(* IEC 61131-3 sources: 2026_Projet_YGO_ExcavatriceDragage/CODE/SIMULATION/PLC_TESTS/SUITE_SAFETY, 3 files *)

(* ---- FB_HeartbeatValidation.st ---- *)
(* ═══════════════════════════════════════════════════════════════
   💓 FB_HeartbeatValidation — Suite table-driven Heartbeat IHM↔PLC
   ───────────────────────────────────────────────────────────────
   📄 Doc : DOC/AF_Partie-14_PLC_Tests_Validation_v1.2.md §7
   🎯 Simulation uniquement. Stimuli amont : toggle IHM, demande SEMI_AUTO,
      retours contacteurs/frein M1/M2, frein M3. Jamais d'écriture dans
      SafeStop/PowerCutOff/HeartbeatOk calculés.
   🧪 TC-H1 sain ; TC-H2 perte 2 s ; TC-H3 reprise sans redémarrage ;
      TC-H4 reset conscient ; TC-H5 escalade Méca B M3.
   ═══════════════════════════════════════════════════════════════ *)

FUNCTION_BLOCK PUBLIC FB_HeartbeatValidation
VAR_INPUT
    Start       : BOOL;
    Abort       : BOOL;
    CaseId      : INT; // 0=tous ; 1..5=cas ciblé
END_VAR
VAR_OUTPUT
    Busy                    : BOOL;
    Done                    : BOOL;
    AnyFailed               : BOOL;
    SimGateOk               : BOOL;
    ActiveStimulusId        : INT;
    StepElapsed             : TIME;
    Report                  : ST_TestSuiteReport;
    TerminalState           : E_TestTerminalState;
    ConfigError             : BOOL;
    ConfigErrorStepId       : INT;
    ConfigErrorCheckIdx     : INT;
    ErrorCode               : INT;
    ErrorMessage            : STRING(160);
END_VAR
VAR CONSTANT
    // ── Sondes ──
    SigHeartbeatIhmOk       : INT := 1;
    SigHeartbeatIhmTimeout  : INT := 2;
    SigSafetyM1ErrorId      : INT := 3;
    SigSafetyM2ErrorId      : INT := 4;
    SigSafetyM3ErrorId      : INT := 5;
    SigCycleErrorId         : INT := 6;
    SigM1FwdRevSpeedFbOff   : INT := 7;
    SigM1BrakeFeedback      : INT := 8;
    SigM2FwdRevSpeedFbOff   : INT := 9;
    SigM2BrakeFeedback      : INT := 10;
    SigM3BrakeFeedback      : INT := 11;
    SigM3DriveActualFreqHz  : INT := 12;
    SigM3DriveStatusWord    : INT := 13;
    SigPowerCutOffActive    : INT := 14;
    // ── Étapes ──
    StepTcH1Setup           : INT := 10;
    StepTcH1WaitToggle      : INT := 11;
    StepTcH1Assert          : INT := 12;
    StepTcH1Teardown        : INT := 19;
    StepTcH2Setup           : INT := 20;
    StepTcH2Freeze          : INT := 21;
    StepTcH2Assert          : INT := 22;
    StepTcH2Teardown        : INT := 29;
    StepTcH3Setup           : INT := 30;
    StepTcH3Resume          : INT := 31;
    StepTcH3Assert          : INT := 32;
    StepTcH3Teardown        : INT := 39;
    StepTcH4Setup           : INT := 40;
    StepTcH4Reset           : INT := 41;
    StepTcH4Assert          : INT := 42;
    StepTcH4Teardown        : INT := 49;
    StepTcH5Setup           : INT := 50;
    StepTcH5MecaB           : INT := 51;
    StepTcH5Assert          : INT := 52;
    StepTcH5Teardown        : INT := 59;
END_VAR
VAR
    // Moteur
    Sequencer               : FB_TestSequencer;
    // Tables
    StepTable               : ARRAY[1..GVL_PLC_Tests_Const.MaxSteps]      OF ST_TestStepConfig;
    CheckTable              : ARRAY[1..GVL_PLC_Tests_Const.MaxChecks]     OF ST_TestCheckConfig;
    CaseTable               : ARRAY[1..GVL_PLC_Tests_Const.MaxTestCases]  OF ST_TestCaseConfig;
    InvariantTable          : ARRAY[1..GVL_PLC_Tests_Const.MaxInvariants] OF ST_TestInvariantConfig;
    // Sondes
    ProbeBool               : ARRAY[1..GVL_PLC_Tests_Const.MaxProbeBool]  OF BOOL;
    ProbeDint               : ARRAY[1..GVL_PLC_Tests_Const.MaxProbeDint]  OF DINT;
    ProbeReal               : ARRAY[1..GVL_PLC_Tests_Const.MaxProbeReal]  OF REAL;
    TableReady              : BOOL := FALSE;
    StartPrev               : BOOL;
    // Stimuli locaux
    StimToggleTimer         : TON;
    StimModeRequest         : E_Mode;
    StimResetPulseTimer     : TON;
END_VAR

// ═══════════════════════════════════════════════════════════════
// 1. 🛡️ GATE
// ═══════════════════════════════════════════════════════════════
IF NOT GVL_Simulation.SimulationModeActive THEN
    Sequencer(Start := FALSE, Abort := TRUE, CaseId := CaseId,
              StepTable := StepTable, CheckTable := CheckTable, CaseTable := CaseTable, InvariantTable := InvariantTable,
              ProbeBool := ProbeBool, ProbeDint := ProbeDint, ProbeReal := ProbeReal, Report := Report);
    GVL_PLC_Tests.OverrideIhmHeartbeatActive := FALSE;
    GVL_PLC_Tests.OverrideM3BrakeStuckOpen := FALSE;
    GVL_PLC_Tests.OverrideM1FwdRevSpeedFbOff := FALSE;
    GVL_PLC_Tests.OverrideM1BrakeFeedback := FALSE;
    GVL_PLC_Tests.OverrideM2FwdRevSpeedFbOff := FALSE;
    GVL_PLC_Tests.OverrideM2BrakeFeedback := FALSE;
    GVL_IHM.Modes.BtnFaultReset := FALSE;
    GVL_IHM.Cycle.CmdReset := FALSE;
    Busy := FALSE; Done := TRUE; AnyFailed := TRUE;
    TerminalState := E_TestTerminalState.TEST_TERMINAL_ABORTED;
    Report.InProgress := FALSE; Report.Aborted := TRUE; Report.AnyFailed := TRUE;
    Report.TerminalState := TerminalState; Report.FailureSummary := 'Heartbeat : NOT SimulationModeActive';
    RETURN;
END_IF;

SimGateOk := GVL_Simulation.SimulationModeActive
          AND NOT GVL_Simulation.SensorM1ContactorFeedbackIsReal
          AND NOT GVL_Simulation.SensorM2ContactorFeedbackIsReal
          AND NOT GVL_Simulation.SensorBrakeThermalIsReal
          AND NOT GVL_Simulation.SensorM3ContactorFeedbackIsReal;

IF Abort OR NOT SimGateOk THEN
    GVL_PLC_Tests.OverrideIhmHeartbeatActive := FALSE;
    GVL_PLC_Tests.OverrideM3BrakeStuckOpen := FALSE;
    GVL_PLC_Tests.OverrideM1FwdRevSpeedFbOff := FALSE;
    GVL_PLC_Tests.OverrideM1BrakeFeedback := FALSE;
    GVL_PLC_Tests.OverrideM2FwdRevSpeedFbOff := FALSE;
    GVL_PLC_Tests.OverrideM2BrakeFeedback := FALSE;
    GVL_IHM.Modes.BtnFaultReset := FALSE;
    GVL_IHM.Cycle.CmdReset := FALSE;
    IF Busy THEN GVL_IHM.Modes.SelMode := StimModeRequest; END_IF;
    Busy := FALSE; Done := TRUE; AnyFailed := TRUE;
    TerminalState := E_TestTerminalState.TEST_TERMINAL_ABORTED;
    Report.InProgress := FALSE; Report.Aborted := TRUE; Report.AnyFailed := TRUE;
    Report.TerminalState := TerminalState; Report.FailureSummary := 'Heartbeat : ABORTED or SimGateOk=FALSE';
    RETURN;
END_IF;

IF Start AND NOT StartPrev AND NOT Busy THEN
    StartPrev := TRUE;
    Busy := TRUE; Done := FALSE; AnyFailed := FALSE; ConfigError := FALSE;
    ErrorCode := 0; ErrorMessage := '';
    StepElapsed := T#0s;
    StimModeRequest := GVL_IHM.Modes.SelMode;

    Report.Name := 'Heartbeat Validation';
    Report.InProgress := TRUE; Report.AllPassed := FALSE; Report.AnyFailed := FALSE; Report.Aborted := FALSE;
    Report.TerminalState := E_TestTerminalState.TEST_TERMINAL_NONE;
    Report.ErrorCode := 0; Report.ErrorMessage := ''; Report.FailureSummary := '';
    Report.FailedTestCase := 0; Report.Duration := T#0s;
    Report.RunCounter := Report.RunCounter + 1;
END_IF;
IF NOT Start THEN StartPrev := FALSE; END_IF;

IF NOT Busy THEN RETURN; END_IF;

// ═══════════════════════════════════════════════════════════════
// 2. 📋 TABLES (remplissage unique)
// ═══════════════════════════════════════════════════════════════
IF NOT TableReady THEN
    Report.Name := 'Heartbeat Validation';

    // ── Cas de tests ──
    CaseTable[1].Name := 'TC-H1 Heartbeat sain';      CaseTable[1].FirstStep := StepTcH1Setup;
    CaseTable[2].Name := 'TC-H2 Perte IHM 2s';        CaseTable[2].FirstStep := StepTcH2Setup;
    CaseTable[3].Name := 'TC-H3 Reprise sans redem';  CaseTable[3].FirstStep := StepTcH3Setup;
    CaseTable[4].Name := 'TC-H4 Reset conscient';     CaseTable[4].FirstStep := StepTcH4Setup;
    CaseTable[5].Name := 'TC-H5 Escalade Meca B M3';  CaseTable[5].FirstStep := StepTcH5Setup;

    // ── Checks (index = ligne CheckTable) ──
    // 1: HeartbeatIhmOk = TRUE
    CheckTable[1].Kind := E_TestCheckKind.BOOL_EQUAL;   CheckTable[1].Mode := E_TestCheckMode.CHECK_WAIT_UNTIL;
    CheckTable[1].ProbeIdx := SigHeartbeatIhmOk;        CheckTable[1].ExpectedBool := TRUE;
    // 2: bit0 Safety M1 = 0
    CheckTable[2].Kind := E_TestCheckKind.WORD_MASK_NONE; CheckTable[2].Mode := E_TestCheckMode.CHECK_WAIT_UNTIL;
    CheckTable[2].ProbeIdx := SigSafetyM1ErrorId;        CheckTable[2].Mask := 16#0001;
    // 3: bit0 Safety M2 = 0
    CheckTable[3].Kind := E_TestCheckKind.WORD_MASK_NONE; CheckTable[3].Mode := E_TestCheckMode.CHECK_WAIT_UNTIL;
    CheckTable[3].ProbeIdx := SigSafetyM2ErrorId;        CheckTable[3].Mask := 16#0001;
    // 4: bit0 Safety M3 = 0
    CheckTable[4].Kind := E_TestCheckKind.WORD_MASK_NONE; CheckTable[4].Mode := E_TestCheckMode.CHECK_WAIT_UNTIL;
    CheckTable[4].ProbeIdx := SigSafetyM3ErrorId;        CheckTable[4].Mask := 16#0001;
    // 5: bit5 Cycle = 0
    CheckTable[5].Kind := E_TestCheckKind.WORD_MASK_NONE; CheckTable[5].Mode := E_TestCheckMode.CHECK_WAIT_UNTIL;
    CheckTable[5].ProbeIdx := SigCycleErrorId;           CheckTable[5].Mask := 16#0020;

    // 6: HeartbeatIhmOk = FALSE
    CheckTable[6].Kind := E_TestCheckKind.BOOL_EQUAL;    CheckTable[6].Mode := E_TestCheckMode.CHECK_WAIT_UNTIL;
    CheckTable[6].ProbeIdx := SigHeartbeatIhmOk;         CheckTable[6].ExpectedBool := FALSE;
    // 7: HeartbeatIhmTimeout = TRUE
    CheckTable[7].Kind := E_TestCheckKind.BOOL_EQUAL;    CheckTable[7].Mode := E_TestCheckMode.CHECK_WAIT_UNTIL;
    CheckTable[7].ProbeIdx := SigHeartbeatIhmTimeout;    CheckTable[7].ExpectedBool := TRUE;
    // 8: bit0 Safety M1 = 1
    CheckTable[8].Kind := E_TestCheckKind.WORD_MASK_ANY; CheckTable[8].Mode := E_TestCheckMode.CHECK_WAIT_UNTIL;
    CheckTable[8].ProbeIdx := SigSafetyM1ErrorId;        CheckTable[8].Mask := 16#0001;
    // 9: bit0 Safety M2 = 1
    CheckTable[9].Kind := E_TestCheckKind.WORD_MASK_ANY; CheckTable[9].Mode := E_TestCheckMode.CHECK_WAIT_UNTIL;
    CheckTable[9].ProbeIdx := SigSafetyM2ErrorId;        CheckTable[9].Mask := 16#0001;
    // 10: bit0 Safety M3 = 1
    CheckTable[10].Kind := E_TestCheckKind.WORD_MASK_ANY; CheckTable[10].Mode := E_TestCheckMode.CHECK_WAIT_UNTIL;
    CheckTable[10].ProbeIdx := SigSafetyM3ErrorId;       CheckTable[10].Mask := 16#0001;
    // 11: bit5 Cycle = 1
    CheckTable[11].Kind := E_TestCheckKind.WORD_MASK_ANY; CheckTable[11].Mode := E_TestCheckMode.CHECK_WAIT_UNTIL;
    CheckTable[11].ProbeIdx := SigCycleErrorId;          CheckTable[11].Mask := 16#0020;

    // 12: SafeStop M1 (via Error)
    CheckTable[12].Kind := E_TestCheckKind.BOOL_EQUAL;   CheckTable[12].Mode := E_TestCheckMode.CHECK_WAIT_UNTIL;
    CheckTable[12].ProbeIdx := SigSafetyM1ErrorId;       CheckTable[12].ExpectedBool := TRUE;
    // 13: SafeStop M2
    CheckTable[13].Kind := E_TestCheckKind.BOOL_EQUAL;   CheckTable[13].Mode := E_TestCheckMode.CHECK_WAIT_UNTIL;
    CheckTable[13].ProbeIdx := SigSafetyM2ErrorId;       CheckTable[13].ExpectedBool := TRUE;
    // 14: SafeStop M3
    CheckTable[14].Kind := E_TestCheckKind.BOOL_EQUAL;   CheckTable[14].Mode := E_TestCheckMode.CHECK_WAIT_UNTIL;
    CheckTable[14].ProbeIdx := SigSafetyM3ErrorId;       CheckTable[14].ExpectedBool := TRUE;

    // 15: HeartbeatIhmOk = TRUE (reprise)
    CheckTable[15].Kind := E_TestCheckKind.BOOL_EQUAL;   CheckTable[15].Mode := E_TestCheckMode.CHECK_WAIT_UNTIL;
    CheckTable[15].ProbeIdx := SigHeartbeatIhmOk;        CheckTable[15].ExpectedBool := TRUE;
    // 16-19: bit0 M1/M2/M3 = 1, bit5 Cycle = 1 (mémorisation)
    CheckTable[16].Kind := E_TestCheckKind.WORD_MASK_ANY; CheckTable[16].Mode := E_TestCheckMode.CHECK_WAIT_UNTIL;
    CheckTable[16].ProbeIdx := SigSafetyM1ErrorId;       CheckTable[16].Mask := 16#0001;
    CheckTable[17].Kind := E_TestCheckKind.WORD_MASK_ANY; CheckTable[17].Mode := E_TestCheckMode.CHECK_WAIT_UNTIL;
    CheckTable[17].ProbeIdx := SigSafetyM2ErrorId;       CheckTable[17].Mask := 16#0001;
    CheckTable[18].Kind := E_TestCheckKind.WORD_MASK_ANY; CheckTable[18].Mode := E_TestCheckMode.CHECK_WAIT_UNTIL;
    CheckTable[18].ProbeIdx := SigSafetyM3ErrorId;       CheckTable[18].Mask := 16#0001;
    CheckTable[19].Kind := E_TestCheckKind.WORD_MASK_ANY; CheckTable[19].Mode := E_TestCheckMode.CHECK_WAIT_UNTIL;
    CheckTable[19].ProbeIdx := SigCycleErrorId;          CheckTable[19].Mask := 16#0020;

    // 20: Reset → bit0 M1/M2/M3 = 0, bit5 Cycle = 0
    CheckTable[20].Kind := E_TestCheckKind.WORD_MASK_NONE; CheckTable[20].Mode := E_TestCheckMode.CHECK_WAIT_UNTIL;
    CheckTable[20].ProbeIdx := SigSafetyM1ErrorId;         CheckTable[20].Mask := 16#0001;
    CheckTable[21].Kind := E_TestCheckKind.WORD_MASK_NONE; CheckTable[21].Mode := E_TestCheckMode.CHECK_WAIT_UNTIL;
    CheckTable[21].ProbeIdx := SigSafetyM2ErrorId;         CheckTable[21].Mask := 16#0001;
    CheckTable[22].Kind := E_TestCheckKind.WORD_MASK_NONE; CheckTable[22].Mode := E_TestCheckMode.CHECK_WAIT_UNTIL;
    CheckTable[22].ProbeIdx := SigSafetyM3ErrorId;         CheckTable[22].Mask := 16#0001;
    CheckTable[23].Kind := E_TestCheckKind.WORD_MASK_NONE; CheckTable[23].Mode := E_TestCheckMode.CHECK_WAIT_UNTIL;
    CheckTable[23].ProbeIdx := SigCycleErrorId;            CheckTable[23].Mask := 16#0020;

    // 24: TC-H5 Méca B M3 — PowerCutOffActive = TRUE
    CheckTable[24].Kind := E_TestCheckKind.BOOL_EQUAL;   CheckTable[24].Mode := E_TestCheckMode.CHECK_WAIT_UNTIL;
    CheckTable[24].ProbeIdx := SigPowerCutOffActive;     CheckTable[24].ExpectedBool := TRUE;

    // ── Étapes ──
    // TC-H1
    StepTable[StepTcH1Setup].Name := 'H1 Setup SEMI_AUTO + toggle sain';
    StepTable[StepTcH1Setup].CaseId := 1; StepTable[StepTcH1Setup].StimulusId := 1;
    StepTable[StepTcH1Setup].CheckIdx[1] := 1; StepTable[StepTcH1Setup].CheckIdx[2] := 2;
    StepTable[StepTcH1Setup].CheckIdx[3] := 3; StepTable[StepTcH1Setup].CheckIdx[4] := 4;
    StepTable[StepTcH1Setup].CheckIdx[5] := 5;
    StepTable[StepTcH1Setup].TimeoutPT := T#5s; StepTable[StepTcH1Setup].NextOnPass := StepTcH1WaitToggle;
    StepTable[StepTcH1Setup].NextOnFail := StepTcH1Teardown; StepTable[StepTcH1Setup].FailAction := E_TestFailAction.FAIL_CONTINUE;

    StepTable[StepTcH1WaitToggle].Name := 'H1 Attente 1er front post-boot';
    StepTable[StepTcH1WaitToggle].CaseId := 1; StepTable[StepTcH1WaitToggle].StimulusId := 1;
    StepTable[StepTcH1WaitToggle].CheckIdx[1] := 1;
    StepTable[StepTcH1WaitToggle].TimeoutPT := T#4s; StepTable[StepTcH1WaitToggle].NextOnPass := StepTcH1Assert;
    StepTable[StepTcH1WaitToggle].NextOnFail := StepTcH1Teardown; StepTable[StepTcH1WaitToggle].FailAction := E_TestFailAction.FAIL_CONTINUE;

    StepTable[StepTcH1Assert].Name := 'H1 Assert bit0=0 & bit5=0';
    StepTable[StepTcH1Assert].CaseId := 1; StepTable[StepTcH1Assert].StimulusId := 1;
    StepTable[StepTcH1Assert].CheckIdx[1] := 2; StepTable[StepTcH1Assert].CheckIdx[2] := 3;
    StepTable[StepTcH1Assert].CheckIdx[3] := 4; StepTable[StepTcH1Assert].CheckIdx[4] := 5;
    StepTable[StepTcH1Assert].TimeoutPT := T#2s; StepTable[StepTcH1Assert].NextOnPass := StepTcH1Teardown;
    StepTable[StepTcH1Assert].NextOnFail := StepTcH1Teardown; StepTable[StepTcH1Assert].FailAction := E_TestFailAction.FAIL_CONTINUE;

    StepTable[StepTcH1Teardown].Name := 'H1 Teardown';
    StepTable[StepTcH1Teardown].CaseId := 1; StepTable[StepTcH1Teardown].StimulusId := 0;
    StepTable[StepTcH1Teardown].DwellPT := T#200ms; StepTable[StepTcH1Teardown].TimeoutPT := T#1s;
    StepTable[StepTcH1Teardown].NextOnPass := 0; StepTable[StepTcH1Teardown].NextOnFail := 0;

    // TC-H2
    StepTable[StepTcH2Setup].Name := 'H2 Setup toggle figé';
    StepTable[StepTcH2Setup].CaseId := 2; StepTable[StepTcH2Setup].StimulusId := 2;
    StepTable[StepTcH2Setup].TimeoutPT := T#1s; StepTable[StepTcH2Setup].NextOnPass := StepTcH2Freeze;
    StepTable[StepTcH2Setup].NextOnFail := StepTcH2Teardown; StepTable[StepTcH2Setup].FailAction := E_TestFailAction.FAIL_CONTINUE;

    StepTable[StepTcH2Freeze].Name := 'H2 Figer toggle > 2s timeout';
    StepTable[StepTcH2Freeze].CaseId := 2; StepTable[StepTcH2Freeze].StimulusId := 2;
    StepTable[StepTcH2Freeze].TimeoutPT := T#3s; StepTable[StepTcH2Freeze].NextOnPass := StepTcH2Assert;
    StepTable[StepTcH2Freeze].NextOnFail := StepTcH2Teardown; StepTable[StepTcH2Freeze].FailAction := E_TestFailAction.FAIL_CONTINUE;

    StepTable[StepTcH2Assert].Name := 'H2 Assert bit0=1 & SafeStop';
    StepTable[StepTcH2Assert].CaseId := 2; StepTable[StepTcH2Assert].StimulusId := 2;
    StepTable[StepTcH2Assert].CheckIdx[1] := 6;  StepTable[StepTcH2Assert].CheckIdx[2] := 7;
    StepTable[StepTcH2Assert].CheckIdx[3] := 8;  StepTable[StepTcH2Assert].CheckIdx[4] := 9;
    StepTable[StepTcH2Assert].CheckIdx[5] := 10; StepTable[StepTcH2Assert].CheckIdx[6] := 11;
    StepTable[StepTcH2Assert].CheckIdx[7] := 12; StepTable[StepTcH2Assert].CheckIdx[8] := 13;
    StepTable[StepTcH2Assert].CheckIdx[9] := 14;
    StepTable[StepTcH2Assert].TimeoutPT := T#3s; StepTable[StepTcH2Assert].NextOnPass := StepTcH2Teardown;
    StepTable[StepTcH2Assert].NextOnFail := StepTcH2Teardown; StepTable[StepTcH2Assert].FailAction := E_TestFailAction.FAIL_CONTINUE;

    StepTable[StepTcH2Teardown].Name := 'H2 Teardown';
    StepTable[StepTcH2Teardown].CaseId := 2; StepTable[StepTcH2Teardown].StimulusId := 0;
    StepTable[StepTcH2Teardown].DwellPT := T#200ms; StepTable[StepTcH2Teardown].TimeoutPT := T#1s;
    StepTable[StepTcH2Teardown].NextOnPass := 0; StepTable[StepTcH2Teardown].NextOnFail := 0;

    // TC-H3
    StepTable[StepTcH3Setup].Name := 'H3 Setup reprise toggle';
    StepTable[StepTcH3Setup].CaseId := 3; StepTable[StepTcH3Setup].StimulusId := 3;
    StepTable[StepTcH3Setup].TimeoutPT := T#1s; StepTable[StepTcH3Setup].NextOnPass := StepTcH3Resume;
    StepTable[StepTcH3Setup].NextOnFail := StepTcH3Teardown; StepTable[StepTcH3Setup].FailAction := E_TestFailAction.FAIL_CONTINUE;

    StepTable[StepTcH3Resume].Name := 'H3 Reprise toggle > 2s';
    StepTable[StepTcH3Resume].CaseId := 3; StepTable[StepTcH3Resume].StimulusId := 3;
    StepTable[StepTcH3Resume].TimeoutPT := T#3s; StepTable[StepTcH3Resume].NextOnPass := StepTcH3Assert;
    StepTable[StepTcH3Resume].NextOnFail := StepTcH3Teardown; StepTable[StepTcH3Resume].FailAction := E_TestFailAction.FAIL_CONTINUE;

    StepTable[StepTcH3Assert].Name := 'H3 Assert bit0=1 & bit5=1';
    StepTable[StepTcH3Assert].CaseId := 3; StepTable[StepTcH3Assert].StimulusId := 3;
    StepTable[StepTcH3Assert].CheckIdx[1] := 15; StepTable[StepTcH3Assert].CheckIdx[2] := 16;
    StepTable[StepTcH3Assert].CheckIdx[3] := 17; StepTable[StepTcH3Assert].CheckIdx[4] := 18;
    StepTable[StepTcH3Assert].CheckIdx[5] := 19;
    StepTable[StepTcH3Assert].TimeoutPT := T#3s; StepTable[StepTcH3Assert].NextOnPass := StepTcH3Teardown;
    StepTable[StepTcH3Assert].NextOnFail := StepTcH3Teardown; StepTable[StepTcH3Assert].FailAction := E_TestFailAction.FAIL_CONTINUE;

    StepTable[StepTcH3Teardown].Name := 'H3 Teardown';
    StepTable[StepTcH3Teardown].CaseId := 3; StepTable[StepTcH3Teardown].StimulusId := 0;
    StepTable[StepTcH3Teardown].DwellPT := T#200ms; StepTable[StepTcH3Teardown].TimeoutPT := T#1s;
    StepTable[StepTcH3Teardown].NextOnPass := 0; StepTable[StepTcH3Teardown].NextOnFail := 0;

    // TC-H4
    StepTable[StepTcH4Setup].Name := 'H4 Setup reset pulse';
    StepTable[StepTcH4Setup].CaseId := 4; StepTable[StepTcH4Setup].StimulusId := 4;
    StepTable[StepTcH4Setup].TimeoutPT := T#1s; StepTable[StepTcH4Setup].NextOnPass := StepTcH4Reset;
    StepTable[StepTcH4Setup].NextOnFail := StepTcH4Teardown; StepTable[StepTcH4Setup].FailAction := E_TestFailAction.FAIL_CONTINUE;

    StepTable[StepTcH4Reset].Name := 'H4 Pulse Reset IHM & Cycle';
    StepTable[StepTcH4Reset].CaseId := 4; StepTable[StepTcH4Reset].StimulusId := 4;
    StepTable[StepTcH4Reset].TimeoutPT := T#2s; StepTable[StepTcH4Reset].NextOnPass := StepTcH4Assert;
    StepTable[StepTcH4Reset].NextOnFail := StepTcH4Teardown; StepTable[StepTcH4Reset].FailAction := E_TestFailAction.FAIL_CONTINUE;

    StepTable[StepTcH4Assert].Name := 'H4 Assert bit0=0 & bit5=0';
    StepTable[StepTcH4Assert].CaseId := 4; StepTable[StepTcH4Assert].StimulusId := 1; // retour toggle sain
    StepTable[StepTcH4Assert].CheckIdx[1] := 20; StepTable[StepTcH4Assert].CheckIdx[2] := 21;
    StepTable[StepTcH4Assert].CheckIdx[3] := 22; StepTable[StepTcH4Assert].CheckIdx[4] := 23;
    StepTable[StepTcH4Assert].TimeoutPT := T#3s; StepTable[StepTcH4Assert].NextOnPass := StepTcH4Teardown;
    StepTable[StepTcH4Assert].NextOnFail := StepTcH4Teardown; StepTable[StepTcH4Assert].FailAction := E_TestFailAction.FAIL_CONTINUE;

    StepTable[StepTcH4Teardown].Name := 'H4 Teardown';
    StepTable[StepTcH4Teardown].CaseId := 4; StepTable[StepTcH4Teardown].StimulusId := 0;
    StepTable[StepTcH4Teardown].DwellPT := T#200ms; StepTable[StepTcH4Teardown].TimeoutPT := T#1s;
    StepTable[StepTcH4Teardown].NextOnPass := 0; StepTable[StepTcH4Teardown].NextOnFail := 0;

    // TC-H5
    StepTable[StepTcH5Setup].Name := 'H5 Setup Meca B M3 frein open';
    StepTable[StepTcH5Setup].CaseId := 5; StepTable[StepTcH5Setup].StimulusId := 5;
    StepTable[StepTcH5Setup].TimeoutPT := T#1s; StepTable[StepTcH5Setup].NextOnPass := StepTcH5MecaB;
    StepTable[StepTcH5Setup].NextOnFail := StepTcH5Teardown; StepTable[StepTcH5Setup].FailAction := E_TestFailAction.FAIL_CONTINUE;

    StepTable[StepTcH5MecaB].Name := 'H5 Perte IHM + M3 open > 3s';
    StepTable[StepTcH5MecaB].CaseId := 5; StepTable[StepTcH5MecaB].StimulusId := 5;
    StepTable[StepTcH5MecaB].TimeoutPT := T#7s; StepTable[StepTcH5MecaB].NextOnPass := StepTcH5Assert;
    StepTable[StepTcH5MecaB].NextOnFail := StepTcH5Teardown; StepTable[StepTcH5MecaB].FailAction := E_TestFailAction.FAIL_CONTINUE;

    StepTable[StepTcH5Assert].Name := 'H5 Assert PowerCutOffActive';
    StepTable[StepTcH5Assert].CaseId := 5; StepTable[StepTcH5Assert].StimulusId := 5;
    StepTable[StepTcH5Assert].CheckIdx[1] := 24;
    StepTable[StepTcH5Assert].TimeoutPT := T#3s; StepTable[StepTcH5Assert].NextOnPass := StepTcH5Teardown;
    StepTable[StepTcH5Assert].NextOnFail := StepTcH5Teardown; StepTable[StepTcH5Assert].FailAction := E_TestFailAction.FAIL_CONTINUE;

    StepTable[StepTcH5Teardown].Name := 'H5 Teardown';
    StepTable[StepTcH5Teardown].CaseId := 5; StepTable[StepTcH5Teardown].StimulusId := 0;
    StepTable[StepTcH5Teardown].DwellPT := T#200ms; StepTable[StepTcH5Teardown].TimeoutPT := T#1s;
    StepTable[StepTcH5Teardown].NextOnPass := 0; StepTable[StepTcH5Teardown].NextOnFail := 0;

    TableReady := TRUE;
END_IF;

// ═══════════════════════════════════════════════════════════════
// 3. 📥 ACQUIRE — câblage sondes (1 ligne par signal, pas de logique)
// ═══════════════════════════════════════════════════════════════
ProbeBool[SigHeartbeatIhmOk]       := PRG_01_Diagnostics.instIhmHeartbeat.HeartbeatIhmOk;
ProbeBool[SigHeartbeatIhmTimeout]  := PRG_01_Diagnostics.instIhmHeartbeat.HeartbeatIhmTimeout;
ProbeDint[SigSafetyM1ErrorId]      := WORD_TO_DINT(PRG_03_Safety.instSafetyWinchM1.ErrorId);
ProbeDint[SigSafetyM2ErrorId]      := WORD_TO_DINT(PRG_03_Safety.instSafetyWinchM2.ErrorId);
ProbeDint[SigSafetyM3ErrorId]      := WORD_TO_DINT(PRG_03_Safety.instSafetyTranslationM3.ErrorId);
ProbeDint[SigCycleErrorId]         := WORD_TO_DINT(PRG_05_Cycle.instCycle.ErrorId);
ProbeBool[SigM1FwdRevSpeedFbOff]   := PRG_00_Inputs.M1FwdRevSpeedFeedbackOff;
ProbeBool[SigM1BrakeFeedback]      := PRG_00_Inputs.M1BrakeFeedback;
ProbeBool[SigM2FwdRevSpeedFbOff]   := PRG_00_Inputs.M2FwdRevSpeedFeedbackOff;
ProbeBool[SigM2BrakeFeedback]      := PRG_00_Inputs.M2BrakeFeedback;
ProbeBool[SigM3BrakeFeedback]      := PRG_00_Inputs.M3BrakeFeedback;
ProbeReal[SigM3DriveActualFreqHz]  := UINT_TO_REAL(PRG_00_Inputs.M3_ActualFrequencyHz_Filtered) / 100.0;
ProbeDint[SigM3DriveStatusWord]    := WORD_TO_DINT(PRG_00_Inputs.M3_StatusWord_Filtered);
ProbeBool[SigPowerCutOffActive]    := GVL_IHM.Modes.PowerCutOffActive;

// ═══════════════════════════════════════════════════════════════
// 4. ⚙️ MOTEUR
// ═══════════════════════════════════════════════════════════════
Sequencer(Start := Start, Abort := Abort, CaseId := CaseId,
          StepTable := StepTable, CheckTable := CheckTable, CaseTable := CaseTable, InvariantTable := InvariantTable,
          ProbeBool := ProbeBool, ProbeDint := ProbeDint, ProbeReal := ProbeReal, Report := Report,
          Busy => Busy, Done => Done, AnyFailed => AnyFailed,
          ConfigError => ConfigError, ConfigErrorStepId => ConfigErrorStepId, ConfigErrorCheckIdx => ConfigErrorCheckIdx,
          ActiveStimulusId => ActiveStimulusId, StepElapsed => StepElapsed,
          TerminalState => TerminalState, ErrorCode => ErrorCode, ErrorMessage => ErrorMessage);

// ═══════════════════════════════════════════════════════════════
// 5. ⚡ STIMULI — modèle hybride : TOR état-complet + pulse timer
// ═══════════════════════════════════════════════════════════════
// StimulusId 0 = neutre garanti (tout relâché) — sur Done/Abort par le moteur
GVL_PLC_Tests.OverrideIhmHeartbeatActive := FALSE;
GVL_PLC_Tests.OverrideM3BrakeStuckOpen := FALSE;
GVL_PLC_Tests.OverrideM1FwdRevSpeedFbOff := FALSE;
GVL_PLC_Tests.OverrideM1BrakeFeedback := FALSE;
GVL_PLC_Tests.OverrideM2FwdRevSpeedFbOff := FALSE;
GVL_PLC_Tests.OverrideM2BrakeFeedback := FALSE;
GVL_IHM.Modes.SelMode := StimModeRequest;
GVL_IHM.Modes.BtnFaultReset := FALSE;
GVL_IHM.Cycle.CmdReset := FALSE;

CASE ActiveStimulusId OF
    1: // TC-H1/TC-H4 : toggle sain 500 ms + SEMI_AUTO
        GVL_PLC_Tests.OverrideIhmHeartbeatActive := TRUE;
        GVL_IHM.Modes.SelMode := E_Mode.SEMI_AUTO;
        // Toggle 500 ms
        StimToggleTimer(IN := TRUE, PT := T#500ms);
        IF StimToggleTimer.Q THEN
            GVL_PLC_Tests.OverrideIhmHeartbeatToggle := NOT GVL_PLC_Tests.OverrideIhmHeartbeatToggle;
            StimToggleTimer(IN := FALSE);
        END_IF;

    2: // TC-H2 : toggle figé (perte IHM)
        GVL_PLC_Tests.OverrideIhmHeartbeatActive := TRUE;
        GVL_IHM.Modes.SelMode := E_Mode.SEMI_AUTO;
        // OverrideIhmHeartbeatToggle figé = pas de front

    3: // TC-H3 : reprise toggle sain
        GVL_PLC_Tests.OverrideIhmHeartbeatActive := TRUE;
        GVL_IHM.Modes.SelMode := E_Mode.SEMI_AUTO;
        StimToggleTimer(IN := TRUE, PT := T#500ms);
        IF StimToggleTimer.Q THEN
            GVL_PLC_Tests.OverrideIhmHeartbeatToggle := NOT GVL_PLC_Tests.OverrideIhmHeartbeatToggle;
            StimToggleTimer(IN := FALSE);
        END_IF;

    4: // TC-H4 : pulse reset conscient
        GVL_PLC_Tests.OverrideIhmHeartbeatActive := TRUE;
        GVL_IHM.Modes.SelMode := E_Mode.SEMI_AUTO;
        StimToggleTimer(IN := TRUE, PT := T#500ms);
        IF StimToggleTimer.Q THEN
            GVL_PLC_Tests.OverrideIhmHeartbeatToggle := NOT GVL_PLC_Tests.OverrideIhmHeartbeatToggle;
            StimToggleTimer(IN := FALSE);
        END_IF;
        StimResetPulseTimer(IN := TRUE, PT := T#1500ms);
        IF NOT StimResetPulseTimer.Q THEN
            GVL_IHM.Modes.BtnFaultReset := TRUE;
            GVL_IHM.Cycle.CmdReset := TRUE;
        END_IF;

    5: // TC-H5 : perte IHM + frein M3 desserré → Méca B
        GVL_PLC_Tests.OverrideIhmHeartbeatActive := TRUE;
        GVL_IHM.Modes.SelMode := E_Mode.SEMI_AUTO;
        GVL_PLC_Tests.OverrideM3BrakeStuckOpen := TRUE; // frein M3 desserré
        // Toggle figé = perte IHM
END_CASE;

// ═══════════════════════════════════════════════════════════════
// 6. 🛑 Premier échec → fin explicite, stimuli relâchés, rapport figé
// ═══════════════════════════════════════════════════════════════
IF ErrorCode <> 0 THEN
    GVL_PLC_Tests.OverrideIhmHeartbeatActive := FALSE;
    GVL_PLC_Tests.OverrideM3BrakeStuckOpen := FALSE;
    GVL_PLC_Tests.OverrideM1FwdRevSpeedFbOff := FALSE;
    GVL_PLC_Tests.OverrideM1BrakeFeedback := FALSE;
    GVL_PLC_Tests.OverrideM2FwdRevSpeedFbOff := FALSE;
    GVL_PLC_Tests.OverrideM2BrakeFeedback := FALSE;
    GVL_IHM.Modes.BtnFaultReset := FALSE;
    GVL_IHM.Cycle.CmdReset := FALSE;
    GVL_IHM.Modes.SelMode := StimModeRequest;
    Busy := FALSE; Done := TRUE; AnyFailed := TRUE;
    TerminalState := E_TestTerminalState.TEST_TERMINAL_FAILED;
    Report.InProgress := FALSE; Report.TerminalState := TerminalState;
END_IF;

(* ---- FB_PLC_Tests_Management.st ---- *)
FUNCTION_BLOCK PUBLIC FB_PLC_Tests_Management
VAR_INPUT
    instBucket                : REFERENCE TO FB_Bucket;     // 🆕 Instance benne (pour FB_BucketValidation)
    instWinchM2               : REFERENCE TO FB_Winch;      // 🆕 Instance treuil M2 (pour FB_BucketValidation)
END_VAR
VAR
    // 🧱 Instances de test (1 par suite — ajouter une suite = 1 instance + 1 branche CASE,
    // voir AF_Partie-14 §7.3.4)
    instSafetyValidation      : FB_SafetyValidation;
    instTranslationValidation : FB_TranslationValidation;
    instBucketValidation      : FB_BucketValidation;
    instEncoderValidation     : FB_EncoderValidation;
    instModesValidation       : FB_ModesValidation;
    instHeartbeatValidation   : FB_HeartbeatValidation;

    // Triggers pour IHM tactiles
    RunAllTrig           : R_TRIG;
    AbortTrig            : R_TRIG;
    ClearReportTrig      : R_TRIG;

    // Variables de commande internes
    StartSafety          : BOOL;
    AbortSafety          : BOOL;
    RequestedCaseSafety  : INT;
    StartTranslation     : BOOL;
    AbortTranslation     : BOOL;
    RequestedCaseTranslation : INT; // 🆕 2026-07-22 : CaseId direct (0=toutes,1..6) — JAMAIS de FirstStepId (audit v1.0 C2)
    StartBucket           : BOOL;
    AbortBucket           : BOOL;
    RequestedCaseBucket   : INT;
    StartEncoder          : BOOL;
    AbortEncoder          : BOOL;
    RequestedCaseEncoder  : INT;
    StartModes            : BOOL;
    AbortModes            : BOOL;
    RequestedCaseModes    : INT;
    StartHeartbeat        : BOOL;
    AbortHeartbeat        : BOOL;
    RequestedCaseHeartbeat : INT;
    StartFramework        : BOOL;
    FrameworkScanCount    : INT;

    // 🔗 Enchaînement multi-suites (CmdRunAll) — 2026-07-16 : ajout Translation puis Bucket
    ChainMode            : BOOL;  // TRUE = run déclenché par RunAll, enchaîne Safety PUIS Translation PUIS Bucket
    CurrentSuiteIdx      : INT;   // Suite active/dernière active (GVL_PLC_Tests_Const.SuiteSafety/SuiteTranslation/SuiteBucket)
    FinalAborted         : BOOL;
    FinalAnyFailed       : BOOL;
    SuiteElapsed         : TIME;
    SuiteWatchdogExpired : BOOL;
    LastLoggedSafetyRun  : UDINT;
    LastLoggedTranslationRun : UDINT;
    LastLoggedBucketRun  : UDINT;
    LastLoggedHeartbeatRun : UDINT;
    EventIdx             : INT;

    // Compteurs pour progression IHM
    Idx                  : INT;
    PassedCount          : INT;
    FailedCount          : INT;
    TotalCount           : INT;

    // 💓 Gestion du clignotant HMI
    LastStepId           : INT := 0;
    PulseCounter         : INT := 0;
    CycleCounter         : INT := 0;
END_VAR
// === IMPLEMENTATION ===
// 1. Détection des commandes HMI
RunAllTrig(CLK := GVL_PLC_Tests.Cmd.RunAll);
AbortTrig(CLK := GVL_PLC_Tests.Cmd.Abort);
ClearReportTrig(CLK := GVL_PLC_Tests.Cmd.ClearReport);

// Remise à zéro des boutons poussoirs HMI
// 🔧 REX 2026-07-16 (demande utilisateur) : CmdRunAll n'est PAS remis à FALSE ici (contrairement
// à l'ancien CmdRunTests, pulse consommé au scan suivant) — il reste TRUE tout le temps du run,
// pratique pour observer en Watch/forçage CODESYS, et ne retombe qu'au Done (cf. CASE ci-dessous).
// R_TRIG garantit qu'un niveau maintenu ne redéclenche pas un 2e run.
IF GVL_PLC_Tests.Cmd.Abort THEN
    GVL_PLC_Tests.Cmd.Abort := FALSE;
END_IF;
IF GVL_PLC_Tests.Cmd.ClearReport THEN
    GVL_PLC_Tests.Cmd.ClearReport := FALSE;
END_IF;

// 2. Machine d'états principale
CASE GVL_PLC_Tests.Status.RunState OF

    // 🔧 REX 2026-07-16 (demande utilisateur) : PASSED/FAILED/ABORTED sont FIGÉS ici (pattern
    // StateAtError, P3 §4) — sans ça, l'état ne durait qu'1 scan (10ms) avant de retomber tout
    // seul à IDLE, invisible en Watch CODESYS. On ne quitte cet état que sur nouveau Start
    // (relance direct un run) ou CmdClearReport (acquittement explicite → retour IDLE).
    E_TestRunState.TESTRUN_IDLE, E_TestRunState.TESTRUN_PASSED, E_TestRunState.TESTRUN_FAILED, E_TestRunState.TESTRUN_ABORTED:
        StartSafety := FALSE;
        AbortSafety := FALSE;
        StartTranslation := FALSE;
        AbortTranslation := FALSE;
        StartBucket := FALSE;
        AbortBucket := FALSE;
        StartEncoder := FALSE;
        AbortEncoder := FALSE;
        StartModes := FALSE;
        AbortModes := FALSE;
        StartHeartbeat := FALSE;
        AbortHeartbeat := FALSE;
        StartFramework := FALSE;
        SuiteElapsed := T#0s;
        SuiteWatchdogExpired := FALSE;

        // 🧪 RunAll prioritaire : démarre une campagne complète depuis Safety.
        IF RunAllTrig.Q THEN
            ChainMode := TRUE;
            CurrentSuiteIdx := GVL_PLC_Tests_Const.SuiteSafety;
            RequestedCaseSafety := 0;
            RequestedCaseTranslation := 0;
            RequestedCaseBucket := 0;
            RequestedCaseEncoder := 0;
            RequestedCaseModes := 0;
            RequestedCaseHeartbeat := 0;
            FinalAborted := FALSE;
            FinalAnyFailed := FALSE;
            GVL_PLC_Tests.Cmd.RunSuite := 0;
            GVL_PLC_Tests.Cmd.RunCase := 0;
            GVL_PLC_Tests.Status.FailureSummary := '';
            StartSafety := TRUE;
            GVL_PLC_Tests.Status.RunState := E_TestRunState.TESTRUN_RUNNING;
        // Normalisation des commandes unitaires vers RunSuite.
        ELSIF GVL_PLC_Tests.Cmd.RunSafety THEN
            GVL_PLC_Tests.Cmd.RunSuite := GVL_PLC_Tests_Const.SuiteSafety;
            GVL_PLC_Tests.Cmd.RunSafety := FALSE;
        ELSIF GVL_PLC_Tests.Cmd.RunTranslation THEN
            GVL_PLC_Tests.Cmd.RunSuite := GVL_PLC_Tests_Const.SuiteTranslation;
            GVL_PLC_Tests.Cmd.RunTranslation := FALSE;
        ELSIF GVL_PLC_Tests.Cmd.RunBucket THEN
            GVL_PLC_Tests.Cmd.RunSuite := GVL_PLC_Tests_Const.SuiteBucket;
            GVL_PLC_Tests.Cmd.RunBucket := FALSE;
        ELSIF GVL_PLC_Tests.Cmd.RunEncoder THEN
            GVL_PLC_Tests.Cmd.RunSuite := GVL_PLC_Tests_Const.SuiteEncoder;
            GVL_PLC_Tests.Cmd.RunEncoder := FALSE;
        ELSIF GVL_PLC_Tests.Cmd.RunModes THEN
            GVL_PLC_Tests.Cmd.RunSuite := GVL_PLC_Tests_Const.SuiteModes;
            GVL_PLC_Tests.Cmd.RunModes := FALSE;
        ELSIF GVL_PLC_Tests.Cmd.RunHeartbeat THEN
            GVL_PLC_Tests.Cmd.RunSuite := GVL_PLC_Tests_Const.SuiteHeartbeat;
            GVL_PLC_Tests.Cmd.RunHeartbeat := FALSE;
        ELSIF GVL_PLC_Tests.Cmd.RunFramework THEN
            StartFramework := TRUE;
            GVL_PLC_Tests.Cmd.RunFramework := FALSE;
        END_IF;

        // Démarrage d'une suite ciblée (Safety)
        IF GVL_PLC_Tests.Cmd.RunSuite = GVL_PLC_Tests_Const.SuiteSafety THEN
            IF GVL_Simulation.SimulationModeActive AND instSafetyValidation.SimGateOk THEN
                ChainMode := FALSE;
                CurrentSuiteIdx := GVL_PLC_Tests_Const.SuiteSafety;
                StartSafety := TRUE;
                RequestedCaseSafety := GVL_PLC_Tests.Cmd.RunCase;
                GVL_PLC_Tests.Status.FailureSummary := ''; // 🔄 RAZ à chaque nouveau run
                GVL_PLC_Tests.Status.RunState := E_TestRunState.TESTRUN_RUNNING;
            END_IF;
            GVL_PLC_Tests.Cmd.RunSuite := 0;
            GVL_PLC_Tests.Cmd.RunCase := 0;

        // Démarrage d'une suite ciblée (Translation)
        // 🆕 2026-07-22 : CaseId transmis TEL QUEL (0=toutes,1..6) — le manager ne
        // connaît plus aucun détail interne d'étape (audit v1.0 C2). Refus de
        // gate désormais explicite PRECONDITION_FAILED, jamais silencieux (C3).
        ELSIF GVL_PLC_Tests.Cmd.RunSuite = GVL_PLC_Tests_Const.SuiteTranslation THEN
            // La suite possède seule sa fixture : même un refus produit un rapport neuf
            // PRECONDITION_FAILED, jamais un Status correct avec un ancien rapport.
            ChainMode := FALSE;
            CurrentSuiteIdx := GVL_PLC_Tests_Const.SuiteTranslation;
            StartTranslation := TRUE;
            RequestedCaseTranslation := GVL_PLC_Tests.Cmd.RunCase;
            GVL_PLC_Tests.Status.FailureSummary := '';
            GVL_PLC_Tests.Status.RunState := E_TestRunState.TESTRUN_RUNNING;
            GVL_PLC_Tests.Cmd.RunSuite := 0;
            GVL_PLC_Tests.Cmd.RunCase := 0;

        // Démarrage d'une suite ciblée (Bucket)
        ELSIF GVL_PLC_Tests.Cmd.RunSuite = GVL_PLC_Tests_Const.SuiteBucket THEN
            IF GVL_Simulation.SimulationModeActive AND instBucketValidation.SimGateOk THEN
                ChainMode := FALSE;
                CurrentSuiteIdx := GVL_PLC_Tests_Const.SuiteBucket;
                StartBucket := TRUE;
                RequestedCaseBucket := GVL_PLC_Tests.Cmd.RunCase;
                GVL_PLC_Tests.Status.FailureSummary := ''; // 🔄 RAZ à chaque nouveau run
                GVL_PLC_Tests.Status.RunState := E_TestRunState.TESTRUN_RUNNING;
            END_IF;
            GVL_PLC_Tests.Cmd.RunSuite := 0;
            GVL_PLC_Tests.Cmd.RunCase := 0;

        // Démarrage d'une suite ciblée (Codeurs/Homing nominal)
        ELSIF GVL_PLC_Tests.Cmd.RunSuite = GVL_PLC_Tests_Const.SuiteEncoder THEN
            IF GVL_Simulation.SimulationModeActive AND instEncoderValidation.SimGateOk THEN
                ChainMode := FALSE;
                CurrentSuiteIdx := GVL_PLC_Tests_Const.SuiteEncoder;
                StartEncoder := TRUE;
                RequestedCaseEncoder := GVL_PLC_Tests.Cmd.RunCase;
                GVL_PLC_Tests.Status.FailureSummary := '';
                GVL_PLC_Tests.Status.RunState := E_TestRunState.TESTRUN_RUNNING;
            END_IF;
            GVL_PLC_Tests.Cmd.RunSuite := 0;
            GVL_PLC_Tests.Cmd.RunCase := 0;

        // Démarrage d'une suite ciblée (Modes/Homme-mort, post-suppression IHM_MANU)
        ELSIF GVL_PLC_Tests.Cmd.RunSuite = GVL_PLC_Tests_Const.SuiteModes THEN
            IF GVL_Simulation.SimulationModeActive AND instModesValidation.SimGateOk THEN
                ChainMode := FALSE;
                CurrentSuiteIdx := GVL_PLC_Tests_Const.SuiteModes;
                StartModes := TRUE;
                RequestedCaseModes := GVL_PLC_Tests.Cmd.RunCase;
                GVL_PLC_Tests.Status.FailureSummary := '';
                GVL_PLC_Tests.Status.RunState := E_TestRunState.TESTRUN_RUNNING;
            END_IF;
            GVL_PLC_Tests.Cmd.RunSuite := 0;
            GVL_PLC_Tests.Cmd.RunCase := 0;

        // Démarrage suite Heartbeat IHM↔PLC.
        ELSIF GVL_PLC_Tests.Cmd.RunSuite = GVL_PLC_Tests_Const.SuiteHeartbeat THEN
            IF GVL_Simulation.SimulationModeActive
               AND NOT GVL_Simulation.SensorM1ContactorFeedbackIsReal
               AND NOT GVL_Simulation.SensorM2ContactorFeedbackIsReal THEN
                ChainMode := FALSE;
                CurrentSuiteIdx := GVL_PLC_Tests_Const.SuiteHeartbeat;
                StartHeartbeat := TRUE;
                RequestedCaseHeartbeat := GVL_PLC_Tests.Cmd.RunCase;
                GVL_PLC_Tests.Status.FailureSummary := '';
                GVL_PLC_Tests.Status.RunState := E_TestRunState.TESTRUN_RUNNING;
            END_IF;
            GVL_PLC_Tests.Cmd.RunSuite := 0;
            GVL_PLC_Tests.Cmd.RunCase := 0;
        END_IF;

        // 🧪 Smoke test géré directement ici : aucune instance/table/runtime.
        IF StartFramework THEN
            ChainMode := FALSE;
            FrameworkScanCount := 0;
            GVL_PLC_Tests.FrameworkResult.InProgress := TRUE;
            GVL_PLC_Tests.FrameworkResult.AllPassed := FALSE;
            GVL_PLC_Tests.FrameworkResult.AnyFailed := FALSE;
            GVL_PLC_Tests.FrameworkResult.CurrentTestId := 1;
            GVL_PLC_Tests.FrameworkResult.FailedTestId := 0;
            GVL_PLC_Tests.FrameworkResult.TestsPassed := 0;
            GVL_PLC_Tests.FrameworkResult.TestsFailed := 0;
            GVL_PLC_Tests.FrameworkResult.ErrorMessage := '';
            GVL_PLC_Tests.FrameworkResult.RunCounter := GVL_PLC_Tests.FrameworkResult.RunCounter + 1;
            GVL_PLC_Tests.Status.FailureSummary := '';
            CurrentSuiteIdx := 7;
            GVL_PLC_Tests.Status.RunState := E_TestRunState.TESTRUN_RUNNING;
        END_IF;

        // Commande d'effacement du rapport — acquittement explicite, retour à IDLE
        IF ClearReportTrig.Q THEN
            // La réinitialisation des rapports Steps[]/Cases[] est gérée par le moteur
            // au démarrage du run suivant ; ici on remet juste les compteurs IHM et on
            // libère l'état figé PASSED/FAILED/ABORTED.
            GVL_PLC_Tests.Status.CasesTotal := 0;
            GVL_PLC_Tests.Status.CasesPassed := 0;
            GVL_PLC_Tests.Status.CasesFailed := 0;
            GVL_PLC_Tests.Status.FailureSummary := '';
            GVL_PLC_Tests.EventCount := 0;
            GVL_PLC_Tests.EventSequence := 0;
            GVL_PLC_Tests.EventOverflow := FALSE;
            GVL_PLC_Tests.Status.RunState := E_TestRunState.TESTRUN_IDLE;
        END_IF;

    E_TestRunState.TESTRUN_RUNNING:
        // Annulation des impulsions de départ
        StartSafety := FALSE;
        StartTranslation := FALSE;
        StartBucket := FALSE;
        StartEncoder := FALSE;
        StartModes := FALSE;
        StartHeartbeat := FALSE;
        StartFramework := FALSE;

        // 🧪 Smoke framework natif : 3 scans, sans appeler aucun moteur de test.
        IF CurrentSuiteIdx = 7 THEN
            FrameworkScanCount := FrameworkScanCount + 1;
            IF FrameworkScanCount >= 3 THEN
                GVL_PLC_Tests.FrameworkResult.InProgress := FALSE;
                GVL_PLC_Tests.FrameworkResult.AllPassed := TRUE;
                GVL_PLC_Tests.FrameworkResult.AnyFailed := FALSE;
                GVL_PLC_Tests.FrameworkResult.TestsPassed := 1;
                GVL_PLC_Tests.FrameworkResult.TestsFailed := 0;
                GVL_PLC_Tests.Status.RunState := E_TestRunState.TESTRUN_PASSED;
            END_IF;
        END_IF;

        // 🛡️ Aucun orchestrateur ne doit attendre Done indéfiniment.
        SuiteElapsed := SuiteElapsed + UDINT_TO_TIME(INT_TO_UDINT(GVL_PLC_Tests_Const.TaskCycleMs));
        GVL_PLC_Tests.Status.SuiteElapsed := SuiteElapsed;
        IF SuiteElapsed >= DINT_TO_TIME(GVL_PLC_Tests_Const.MaxSuiteDurationMs) THEN
            SuiteWatchdogExpired := TRUE;
            GVL_PLC_Tests.Status.SuiteWatchdogExpired := TRUE;
            IF CurrentSuiteIdx = GVL_PLC_Tests_Const.SuiteSafety THEN
                AbortSafety := TRUE;
            ELSIF CurrentSuiteIdx = GVL_PLC_Tests_Const.SuiteTranslation THEN
                AbortTranslation := TRUE;
            ELSIF CurrentSuiteIdx = GVL_PLC_Tests_Const.SuiteEncoder THEN
                AbortEncoder := TRUE;
            ELSIF CurrentSuiteIdx = GVL_PLC_Tests_Const.SuiteModes THEN
                AbortModes := TRUE;
            ELSIF CurrentSuiteIdx = GVL_PLC_Tests_Const.SuiteHeartbeat THEN
                AbortHeartbeat := TRUE;
            ELSE
                AbortBucket := TRUE;
            END_IF;
        END_IF;

        // Abandon propre ou perte du mode Simulation — coupe la suite active
        IF AbortTrig.Q OR NOT GVL_Simulation.SimulationModeActive THEN
            AbortSafety := TRUE;
            AbortTranslation := TRUE;
            AbortBucket := TRUE;
            AbortEncoder := TRUE;
            AbortModes := TRUE;
            AbortHeartbeat := TRUE;
        END_IF;

        // Surveillance de la fin d'exécution — Safety d'abord
        IF CurrentSuiteIdx = GVL_PLC_Tests_Const.SuiteSafety AND instSafetyValidation.Done THEN
            AbortSafety := FALSE;
            IF instSafetyValidation.TerminalState <> E_TestTerminalState.TEST_TERMINAL_DONE AND instSafetyValidation.Report.RunCounter <> LastLoggedSafetyRun THEN
                LastLoggedSafetyRun := instSafetyValidation.Report.RunCounter;
                GVL_PLC_Tests.EventSequence := GVL_PLC_Tests.EventSequence + 1;
                IF GVL_PLC_Tests.EventCount < GVL_PLC_Tests_Const.MaxTestEvents THEN
                    GVL_PLC_Tests.EventCount := GVL_PLC_Tests.EventCount + 1;
                ELSE
                    GVL_PLC_Tests.EventOverflow := TRUE;
                END_IF;
                EventIdx := UDINT_TO_INT(GVL_PLC_Tests.EventSequence MOD INT_TO_UDINT(GVL_PLC_Tests_Const.MaxTestEvents)) + 1;
                GVL_PLC_Tests.EventLog[EventIdx].Sequence := GVL_PLC_Tests.EventSequence;
                GVL_PLC_Tests.EventLog[EventIdx].Severity := E_TestEventSeverity.TEST_EVENT_ERROR;
                GVL_PLC_Tests.EventLog[EventIdx].SuiteId := GVL_PLC_Tests_Const.SuiteSafety;
                GVL_PLC_Tests.EventLog[EventIdx].CaseId := instSafetyValidation.Report.CurrentCaseId;
                GVL_PLC_Tests.EventLog[EventIdx].StepId := instSafetyValidation.Report.CurrentStepId;
                GVL_PLC_Tests.EventLog[EventIdx].Code := instSafetyValidation.ErrorCode;
                GVL_PLC_Tests.EventLog[EventIdx].Message := instSafetyValidation.ErrorMessage;
            END_IF;
            IF ChainMode AND (NOT instSafetyValidation.Report.Aborted OR SuiteWatchdogExpired) AND instTranslationValidation.SimGateOk THEN
                // 🔗 Enchaîne vers Translation (continue même si Safety a échoué — logique
                // FAIL_CONTINUE déjà appliquée au niveau des cases/steps, voir §7.3.4)
                CurrentSuiteIdx := GVL_PLC_Tests_Const.SuiteTranslation;
                SuiteElapsed := T#0s;
                StartTranslation := TRUE;
                RequestedCaseTranslation := 0; // Enchaînement RunAll -> toutes les cases Translation
            ELSIF ChainMode AND NOT instSafetyValidation.Report.Aborted AND NOT instTranslationValidation.SimGateOk THEN
                // 🔧 REX 2026-07-16 : bug trouvé — le chaînage sautait la vérification SimGateOk
                // (le démarrage ciblé Cmd.RunSuite=2 la faisait, pas celui-ci). Sans ce garde-fou,
                // Translation démarrait quand même avec FB_Safety_Translation.Enable=FALSE
                // (ManuActive actif) → 3 timeouts silencieux, aucun défaut jamais détectable.
                GVL_PLC_Tests.Cmd.RunAll := FALSE;
                ChainMode := FALSE; // 🔒 Évite d'agréger un rapport Translation périmé (suite jamais lancée ce run)
                IF instSafetyValidation.Report.FailureSummary = '' THEN
                    GVL_PLC_Tests.Status.FailureSummary := 'Translation NON TESTEE (SimGateOk=FALSE — vérifier SimulationModeActive et les E/S M3 non réelles)';
                ELSE
                    GVL_PLC_Tests.Status.FailureSummary := CONCAT(instSafetyValidation.Report.FailureSummary, ' || Translation NON TESTEE (SimGateOk=FALSE — vérifier SimulationModeActive et les E/S M3 non réelles)');
                END_IF;
                GVL_PLC_Tests.Status.RunState := E_TestRunState.TESTRUN_ABORTED;
            ELSE
                FinalAborted := instSafetyValidation.Report.Aborted;
                FinalAnyFailed := instSafetyValidation.AnyFailed;
                GVL_PLC_Tests.Cmd.RunAll := FALSE; // 🔧 Retombe ICI (Done atteint), pas au démarrage
                GVL_PLC_Tests.Status.FailureSummary := instSafetyValidation.Report.FailureSummary;
                IF FinalAborted THEN
                    GVL_PLC_Tests.Status.RunState := E_TestRunState.TESTRUN_ABORTED;
                ELSIF FinalAnyFailed THEN
                    GVL_PLC_Tests.Status.RunState := E_TestRunState.TESTRUN_FAILED;
                ELSE
                    GVL_PLC_Tests.Status.RunState := E_TestRunState.TESTRUN_PASSED;
                END_IF;
            END_IF;

        // Surveillance de la fin d'exécution — Translation (ciblée ou enchaînée après Safety)
        ELSIF CurrentSuiteIdx = GVL_PLC_Tests_Const.SuiteTranslation AND instTranslationValidation.Done THEN
            AbortTranslation := FALSE;
            IF instTranslationValidation.TerminalState <> E_TestTerminalState.TEST_TERMINAL_DONE AND instTranslationValidation.Report.RunCounter <> LastLoggedTranslationRun THEN
                LastLoggedTranslationRun := instTranslationValidation.Report.RunCounter;
                GVL_PLC_Tests.EventSequence := GVL_PLC_Tests.EventSequence + 1;
                IF GVL_PLC_Tests.EventCount < GVL_PLC_Tests_Const.MaxTestEvents THEN
                    GVL_PLC_Tests.EventCount := GVL_PLC_Tests.EventCount + 1;
                ELSE
                    GVL_PLC_Tests.EventOverflow := TRUE;
                END_IF;
                EventIdx := UDINT_TO_INT(GVL_PLC_Tests.EventSequence MOD INT_TO_UDINT(GVL_PLC_Tests_Const.MaxTestEvents)) + 1;
                GVL_PLC_Tests.EventLog[EventIdx].Sequence := GVL_PLC_Tests.EventSequence;
                GVL_PLC_Tests.EventLog[EventIdx].Severity := E_TestEventSeverity.TEST_EVENT_ERROR;
                GVL_PLC_Tests.EventLog[EventIdx].SuiteId := GVL_PLC_Tests_Const.SuiteTranslation;
                GVL_PLC_Tests.EventLog[EventIdx].CaseId := instTranslationValidation.Report.CurrentCaseId;
                GVL_PLC_Tests.EventLog[EventIdx].StepId := instTranslationValidation.Report.CurrentStepId;
                GVL_PLC_Tests.EventLog[EventIdx].Code := instTranslationValidation.ErrorCode;
                GVL_PLC_Tests.EventLog[EventIdx].Message := instTranslationValidation.ErrorMessage;
            END_IF;
            IF ChainMode AND (NOT instTranslationValidation.Report.Aborted OR SuiteWatchdogExpired) AND instBucketValidation.SimGateOk THEN
                // 🔗 Enchaîne vers Bucket (2026-07-16 : 3e maillon Safety→Translation→Bucket)
                CurrentSuiteIdx := GVL_PLC_Tests_Const.SuiteBucket;
                SuiteElapsed := T#0s;
                StartBucket := TRUE;
                RequestedCaseBucket := 0;
            ELSIF ChainMode AND NOT instTranslationValidation.Report.Aborted AND NOT instBucketValidation.SimGateOk THEN
                // Même garde-fou que Safety→Translation : Bucket ne doit jamais démarrer sans son
                // SimGateOk (refuse si M1/M2 en simulation réelle, voir FB_BucketValidation §1).
                GVL_PLC_Tests.Cmd.RunAll := FALSE;
                ChainMode := FALSE; // 🔒 Évite d'agréger un rapport Bucket périmé (suite jamais lancée ce run)
                IF instSafetyValidation.Report.FailureSummary = '' AND instTranslationValidation.Report.FailureSummary = '' THEN
                    GVL_PLC_Tests.Status.FailureSummary := 'Bucket NON TESTEE (SimGateOk=FALSE — verifier simulation reelle M1/M2)';
                ELSIF instTranslationValidation.Report.FailureSummary = '' THEN
                    GVL_PLC_Tests.Status.FailureSummary := CONCAT(instSafetyValidation.Report.FailureSummary, ' || Bucket NON TESTEE (SimGateOk=FALSE — verifier simulation reelle M1/M2)');
                ELSE
                    GVL_PLC_Tests.Status.FailureSummary := CONCAT(instTranslationValidation.Report.FailureSummary, ' || Bucket NON TESTEE (SimGateOk=FALSE — verifier simulation reelle M1/M2)');
                END_IF;
                GVL_PLC_Tests.Status.RunState := E_TestRunState.TESTRUN_ABORTED;
            ELSE
                // Soit run ciblé (pas de chaînage), soit chaînage interrompu (Translation.Aborted)
                IF ChainMode THEN
                    FinalAborted := instSafetyValidation.Report.Aborted OR instTranslationValidation.Report.Aborted;
                    FinalAnyFailed := instSafetyValidation.AnyFailed OR instTranslationValidation.AnyFailed;
                    IF instSafetyValidation.Report.FailureSummary <> '' AND instTranslationValidation.Report.FailureSummary <> '' THEN
                        GVL_PLC_Tests.Status.FailureSummary := CONCAT(instSafetyValidation.Report.FailureSummary, CONCAT(' || ', instTranslationValidation.Report.FailureSummary));
                    ELSIF instSafetyValidation.Report.FailureSummary <> '' THEN
                        GVL_PLC_Tests.Status.FailureSummary := instSafetyValidation.Report.FailureSummary;
                    ELSE
                        GVL_PLC_Tests.Status.FailureSummary := instTranslationValidation.Report.FailureSummary;
                    END_IF;
                ELSE
                    FinalAborted := instTranslationValidation.Report.Aborted;
                    FinalAnyFailed := instTranslationValidation.AnyFailed;
                    GVL_PLC_Tests.Status.FailureSummary := instTranslationValidation.Report.FailureSummary;
                END_IF;
                GVL_PLC_Tests.Cmd.RunAll := FALSE; // 🔧 Retombe ICI (Done atteint), pas au démarrage
                IF FinalAborted THEN
                    GVL_PLC_Tests.Status.RunState := E_TestRunState.TESTRUN_ABORTED;
                ELSIF FinalAnyFailed THEN
                    GVL_PLC_Tests.Status.RunState := E_TestRunState.TESTRUN_FAILED;
                ELSE
                    GVL_PLC_Tests.Status.RunState := E_TestRunState.TESTRUN_PASSED;
                END_IF;
            END_IF;

        // Surveillance de la fin d'exécution — Bucket (ciblée, ou dernier maillon de la chaîne)
        ELSIF CurrentSuiteIdx = GVL_PLC_Tests_Const.SuiteBucket AND instBucketValidation.Done THEN
            AbortBucket := FALSE;
            IF instBucketValidation.TerminalState <> E_TestTerminalState.TEST_TERMINAL_DONE AND instBucketValidation.Report.RunCounter <> LastLoggedBucketRun THEN
                LastLoggedBucketRun := instBucketValidation.Report.RunCounter;
                GVL_PLC_Tests.EventSequence := GVL_PLC_Tests.EventSequence + 1;
                IF GVL_PLC_Tests.EventCount < GVL_PLC_Tests_Const.MaxTestEvents THEN
                    GVL_PLC_Tests.EventCount := GVL_PLC_Tests.EventCount + 1;
                ELSE
                    GVL_PLC_Tests.EventOverflow := TRUE;
                END_IF;
                EventIdx := UDINT_TO_INT(GVL_PLC_Tests.EventSequence MOD INT_TO_UDINT(GVL_PLC_Tests_Const.MaxTestEvents)) + 1;
                GVL_PLC_Tests.EventLog[EventIdx].Sequence := GVL_PLC_Tests.EventSequence;
                GVL_PLC_Tests.EventLog[EventIdx].Severity := E_TestEventSeverity.TEST_EVENT_ERROR;
                GVL_PLC_Tests.EventLog[EventIdx].SuiteId := GVL_PLC_Tests_Const.SuiteBucket;
                GVL_PLC_Tests.EventLog[EventIdx].CaseId := instBucketValidation.Report.CurrentCaseId;
                GVL_PLC_Tests.EventLog[EventIdx].StepId := instBucketValidation.Report.CurrentStepId;
                GVL_PLC_Tests.EventLog[EventIdx].Code := instBucketValidation.ErrorCode;
                GVL_PLC_Tests.EventLog[EventIdx].Message := instBucketValidation.ErrorMessage;
            END_IF;
            IF ChainMode THEN
                // Campagne complète : Bucket terminé → Encoder.
                CurrentSuiteIdx := GVL_PLC_Tests_Const.SuiteEncoder;
                SuiteElapsed := T#0s;
                StartEncoder := TRUE;
                RequestedCaseEncoder := 0;
                // Conserve les verdicts précédents pour le verdict final.
                FinalAborted := FinalAborted OR instSafetyValidation.Report.Aborted OR instTranslationValidation.Report.Aborted OR instBucketValidation.Report.Aborted;
                FinalAnyFailed := FinalAnyFailed OR instSafetyValidation.AnyFailed OR instTranslationValidation.AnyFailed OR instBucketValidation.AnyFailed;
                // 🏷️ Combine jusqu'à 3 résumés intermédiaires.
                GVL_PLC_Tests.Status.FailureSummary := '';
                IF instSafetyValidation.Report.FailureSummary <> '' THEN
                    GVL_PLC_Tests.Status.FailureSummary := instSafetyValidation.Report.FailureSummary;
                END_IF;
                IF instTranslationValidation.Report.FailureSummary <> '' THEN
                    IF GVL_PLC_Tests.Status.FailureSummary <> '' THEN
                        GVL_PLC_Tests.Status.FailureSummary := CONCAT(GVL_PLC_Tests.Status.FailureSummary, CONCAT(' || ', instTranslationValidation.Report.FailureSummary));
                    ELSE
                        GVL_PLC_Tests.Status.FailureSummary := instTranslationValidation.Report.FailureSummary;
                    END_IF;
                END_IF;
                IF instBucketValidation.Report.FailureSummary <> '' THEN
                    IF GVL_PLC_Tests.Status.FailureSummary <> '' THEN
                        GVL_PLC_Tests.Status.FailureSummary := CONCAT(GVL_PLC_Tests.Status.FailureSummary, CONCAT(' || ', instBucketValidation.Report.FailureSummary));
                    ELSE
                        GVL_PLC_Tests.Status.FailureSummary := instBucketValidation.Report.FailureSummary;
                    END_IF;
                END_IF;
            ELSE
                FinalAborted := instBucketValidation.Report.Aborted;
                FinalAnyFailed := instBucketValidation.AnyFailed;
                GVL_PLC_Tests.Status.FailureSummary := instBucketValidation.Report.FailureSummary;
                GVL_PLC_Tests.Cmd.RunAll := FALSE;
                IF FinalAborted THEN
                    GVL_PLC_Tests.Status.RunState := E_TestRunState.TESTRUN_ABORTED;
                ELSIF FinalAnyFailed THEN
                    GVL_PLC_Tests.Status.RunState := E_TestRunState.TESTRUN_FAILED;
                ELSE
                    GVL_PLC_Tests.Status.RunState := E_TestRunState.TESTRUN_PASSED;
                END_IF;
            END_IF;
        ELSIF CurrentSuiteIdx = GVL_PLC_Tests_Const.SuiteHeartbeat AND instHeartbeatValidation.Done THEN
            AbortHeartbeat := FALSE;
            FinalAborted := FinalAborted OR instHeartbeatValidation.Report.Aborted;
            FinalAnyFailed := FinalAnyFailed OR instHeartbeatValidation.AnyFailed;
            IF instHeartbeatValidation.Report.FailureSummary <> '' THEN
                IF GVL_PLC_Tests.Status.FailureSummary <> '' THEN
                    GVL_PLC_Tests.Status.FailureSummary := CONCAT(GVL_PLC_Tests.Status.FailureSummary, CONCAT(' || ', instHeartbeatValidation.Report.FailureSummary));
                ELSE
                    GVL_PLC_Tests.Status.FailureSummary := instHeartbeatValidation.Report.FailureSummary;
                END_IF;
            END_IF;
            // ChainMode reste mémorisé au terminal pour agréger toute la campagne.
            // Le prochain lancement ciblé le remet explicitement à FALSE.
            GVL_PLC_Tests.Cmd.RunAll := FALSE;
            IF FinalAborted THEN
                GVL_PLC_Tests.Status.RunState := E_TestRunState.TESTRUN_ABORTED;
            ELSIF FinalAnyFailed THEN
                GVL_PLC_Tests.Status.RunState := E_TestRunState.TESTRUN_FAILED;
            ELSE
                GVL_PLC_Tests.Status.RunState := E_TestRunState.TESTRUN_PASSED;
            END_IF;
        ELSIF CurrentSuiteIdx = GVL_PLC_Tests_Const.SuiteEncoder AND instEncoderValidation.Done THEN
            AbortEncoder := FALSE;
            IF ChainMode THEN
                FinalAborted := FinalAborted OR instEncoderValidation.Report.Aborted;
                FinalAnyFailed := FinalAnyFailed OR instEncoderValidation.AnyFailed;
                IF instEncoderValidation.Report.FailureSummary <> '' THEN
                    IF GVL_PLC_Tests.Status.FailureSummary <> '' THEN
                        GVL_PLC_Tests.Status.FailureSummary := CONCAT(GVL_PLC_Tests.Status.FailureSummary, CONCAT(' || ', instEncoderValidation.Report.FailureSummary));
                    ELSE
                        GVL_PLC_Tests.Status.FailureSummary := instEncoderValidation.Report.FailureSummary;
                    END_IF;
                END_IF;
                CurrentSuiteIdx := GVL_PLC_Tests_Const.SuiteModes;
                SuiteElapsed := T#0s;
                StartModes := TRUE;
                RequestedCaseModes := 0;
            ELSE
                FinalAborted := instEncoderValidation.Report.Aborted;
                FinalAnyFailed := instEncoderValidation.AnyFailed;
                GVL_PLC_Tests.Status.FailureSummary := instEncoderValidation.Report.FailureSummary;
            END_IF;
            IF SuiteWatchdogExpired THEN
                GVL_PLC_Tests.Status.FailureSummary := 'Watchdog suite Encoder/Homing expire';
                FinalAborted := FALSE;
                FinalAnyFailed := TRUE;
            END_IF;
            IF NOT ChainMode THEN
                IF FinalAborted THEN
                    GVL_PLC_Tests.Status.RunState := E_TestRunState.TESTRUN_ABORTED;
                ELSIF FinalAnyFailed THEN
                    GVL_PLC_Tests.Status.RunState := E_TestRunState.TESTRUN_FAILED;
                ELSE
                    GVL_PLC_Tests.Status.RunState := E_TestRunState.TESTRUN_PASSED;
                END_IF;
            END_IF;
        ELSIF CurrentSuiteIdx = GVL_PLC_Tests_Const.SuiteModes AND instModesValidation.Done THEN
            AbortModes := FALSE;
            IF ChainMode THEN
                FinalAborted := FinalAborted OR instModesValidation.Report.Aborted;
                FinalAnyFailed := FinalAnyFailed OR instModesValidation.AnyFailed;
                IF instModesValidation.Report.FailureSummary <> '' THEN
                    IF GVL_PLC_Tests.Status.FailureSummary <> '' THEN
                        GVL_PLC_Tests.Status.FailureSummary := CONCAT(GVL_PLC_Tests.Status.FailureSummary, CONCAT(' || ', instModesValidation.Report.FailureSummary));
                    ELSE
                        GVL_PLC_Tests.Status.FailureSummary := instModesValidation.Report.FailureSummary;
                    END_IF;
                END_IF;
                CurrentSuiteIdx := GVL_PLC_Tests_Const.SuiteHeartbeat;
                SuiteElapsed := T#0s;
                StartHeartbeat := TRUE;
                RequestedCaseHeartbeat := 0;
            ELSE
                FinalAborted := instModesValidation.Report.Aborted;
                FinalAnyFailed := instModesValidation.AnyFailed;
                GVL_PLC_Tests.Status.FailureSummary := instModesValidation.Report.FailureSummary;
            END_IF;
            IF SuiteWatchdogExpired THEN
                GVL_PLC_Tests.Status.FailureSummary := 'Watchdog suite Modes/Homme-mort expire';
                FinalAborted := FALSE;
                FinalAnyFailed := TRUE;
            END_IF;
            IF NOT ChainMode THEN
                IF FinalAborted THEN
                    GVL_PLC_Tests.Status.RunState := E_TestRunState.TESTRUN_ABORTED;
                ELSIF FinalAnyFailed THEN
                    GVL_PLC_Tests.Status.RunState := E_TestRunState.TESTRUN_FAILED;
                ELSE
                    GVL_PLC_Tests.Status.RunState := E_TestRunState.TESTRUN_PASSED;
                END_IF;
            END_IF;
        END_IF;

END_CASE;

// 3. Appel des instances de suites
instSafetyValidation(Start := StartSafety, Abort := AbortSafety, CaseId := RequestedCaseSafety);
instTranslationValidation(Start := StartTranslation, Abort := AbortTranslation, CaseId := RequestedCaseTranslation);
instBucketValidation(Start := StartBucket, Abort := AbortBucket, CaseId := RequestedCaseBucket, instBucket := instBucket, instWinchM2 := instWinchM2);
instEncoderValidation(Start := StartEncoder, Abort := AbortEncoder, CaseId := RequestedCaseEncoder);
instModesValidation(Start := StartModes, Abort := AbortModes, CaseId := RequestedCaseModes);
instHeartbeatValidation(Start := StartHeartbeat, Abort := AbortHeartbeat, CaseId := RequestedCaseHeartbeat);

// 4. Centralisation et recopie vers GVL_PLC_Tests
GVL_PLC_Tests.Status.SimulationActive := GVL_Simulation.SimulationModeActive;
GVL_PLC_Tests.Status.SuiteWatchdogExpired := SuiteWatchdogExpired;
GVL_PLC_Tests.SuiteSafetyValidation := instSafetyValidation.Report;
GVL_PLC_Tests.SuiteTranslationValidation := instTranslationValidation.Report;
GVL_PLC_Tests.SuiteTranslationResult := instTranslationValidation.Result; // 🆕 Résultat plat clair
GVL_PLC_Tests.SuiteBucketValidation := instBucketValidation.Report;
GVL_PLC_Tests.SuiteEncoderValidation := instEncoderValidation.Report;
GVL_PLC_Tests.SuiteModesValidation := instModesValidation.Report;
GVL_PLC_Tests.SuiteHeartbeatValidation := instHeartbeatValidation.Report;

// 5. Mise à jour des indicateurs de progression IHM
IF GVL_PLC_Tests.Status.RunState = E_TestRunState.TESTRUN_RUNNING THEN
    GVL_PLC_Tests.Status.ActiveSuiteId := CurrentSuiteIdx;
    // 🧪 L'autotest framework a sa propre progression : ne jamais afficher
    // le rapport Safety résiduel lorsque CurrentSuiteIdx=7.
    IF CurrentSuiteIdx = 7 THEN
        GVL_PLC_Tests.Status.ActiveSuiteName := 'Framework Validation';
        GVL_PLC_Tests.Status.ActiveCaseId := GVL_PLC_Tests.FrameworkResult.CurrentTestId;
        GVL_PLC_Tests.Status.ActiveStepId := GVL_PLC_Tests.FrameworkResult.CurrentTestId;
        GVL_PLC_Tests.Status.StepElapsed := T#0s;
        GVL_PLC_Tests.Status.TerminalState := E_TestTerminalState.TEST_TERMINAL_NONE;
        GVL_PLC_Tests.Status.ErrorCode := GVL_PLC_Tests.FrameworkResult.FailedTestId;
        GVL_PLC_Tests.Status.ErrorMessage := GVL_PLC_Tests.FrameworkResult.ErrorMessage;
    ELSIF CurrentSuiteIdx = GVL_PLC_Tests_Const.SuiteTranslation THEN
        GVL_PLC_Tests.Status.ActiveSuiteName := instTranslationValidation.Report.Name;
        GVL_PLC_Tests.Status.ActiveCaseId := instTranslationValidation.Report.CurrentCaseId;
        GVL_PLC_Tests.Status.ActiveStepId := instTranslationValidation.Report.CurrentStepId;
        GVL_PLC_Tests.Status.StepElapsed := instTranslationValidation.StepElapsed;
        GVL_PLC_Tests.Status.TerminalState := instTranslationValidation.TerminalState;
        GVL_PLC_Tests.Status.ErrorCode := instTranslationValidation.ErrorCode;
        GVL_PLC_Tests.Status.ErrorMessage := instTranslationValidation.ErrorMessage;
    ELSIF CurrentSuiteIdx = GVL_PLC_Tests_Const.SuiteBucket THEN
        GVL_PLC_Tests.Status.ActiveSuiteName := instBucketValidation.Report.Name;
        GVL_PLC_Tests.Status.ActiveCaseId := instBucketValidation.Report.CurrentCaseId;
        GVL_PLC_Tests.Status.ActiveStepId := instBucketValidation.Report.CurrentStepId;
        GVL_PLC_Tests.Status.StepElapsed := instBucketValidation.StepElapsed;
        GVL_PLC_Tests.Status.TerminalState := instBucketValidation.TerminalState;
        GVL_PLC_Tests.Status.ErrorCode := instBucketValidation.ErrorCode;
        GVL_PLC_Tests.Status.ErrorMessage := instBucketValidation.ErrorMessage;
    ELSIF CurrentSuiteIdx = GVL_PLC_Tests_Const.SuiteEncoder THEN
        GVL_PLC_Tests.Status.ActiveSuiteName := instEncoderValidation.Report.Name;
        GVL_PLC_Tests.Status.ActiveCaseId := instEncoderValidation.Report.CurrentCaseId;
        GVL_PLC_Tests.Status.ActiveStepId := instEncoderValidation.Report.CurrentStepId;
        GVL_PLC_Tests.Status.StepElapsed := instEncoderValidation.StepElapsed;
        GVL_PLC_Tests.Status.TerminalState := instEncoderValidation.TerminalState;
        GVL_PLC_Tests.Status.ErrorCode := instEncoderValidation.ErrorCode;
        GVL_PLC_Tests.Status.ErrorMessage := instEncoderValidation.ErrorMessage;
    ELSIF CurrentSuiteIdx = GVL_PLC_Tests_Const.SuiteHeartbeat THEN
        GVL_PLC_Tests.Status.ActiveSuiteName := instHeartbeatValidation.Report.Name;
        GVL_PLC_Tests.Status.ActiveCaseId := instHeartbeatValidation.Report.CurrentCaseId;
        GVL_PLC_Tests.Status.ActiveStepId := instHeartbeatValidation.Report.CurrentStepId;
        GVL_PLC_Tests.Status.StepElapsed := instHeartbeatValidation.StepElapsed;
        GVL_PLC_Tests.Status.TerminalState := instHeartbeatValidation.TerminalState;
        GVL_PLC_Tests.Status.ErrorCode := instHeartbeatValidation.ErrorCode;
        GVL_PLC_Tests.Status.ErrorMessage := instHeartbeatValidation.ErrorMessage;
    ELSIF CurrentSuiteIdx = GVL_PLC_Tests_Const.SuiteModes THEN
        GVL_PLC_Tests.Status.ActiveSuiteName := instModesValidation.Report.Name;
        GVL_PLC_Tests.Status.ActiveCaseId := instModesValidation.Report.CurrentCaseId;
        GVL_PLC_Tests.Status.ActiveStepId := instModesValidation.Report.CurrentStepId;
        GVL_PLC_Tests.Status.StepElapsed := instModesValidation.StepElapsed;
        GVL_PLC_Tests.Status.TerminalState := instModesValidation.TerminalState;
        GVL_PLC_Tests.Status.ErrorCode := instModesValidation.ErrorCode;
        GVL_PLC_Tests.Status.ErrorMessage := instModesValidation.ErrorMessage;
    ELSE
        GVL_PLC_Tests.Status.ActiveSuiteName := instSafetyValidation.Report.Name;
        GVL_PLC_Tests.Status.ActiveCaseId := instSafetyValidation.Report.CurrentCaseId;
        GVL_PLC_Tests.Status.ActiveStepId := instSafetyValidation.Report.CurrentStepId;
        GVL_PLC_Tests.Status.StepElapsed := instSafetyValidation.StepElapsed;
        GVL_PLC_Tests.Status.TerminalState := instSafetyValidation.TerminalState;
        GVL_PLC_Tests.Status.ErrorCode := instSafetyValidation.ErrorCode;
        GVL_PLC_Tests.Status.ErrorMessage := instSafetyValidation.ErrorMessage;
    END_IF;
ELSE
    GVL_PLC_Tests.Status.ActiveSuiteId := 0;
    GVL_PLC_Tests.Status.ActiveSuiteName := '';
    GVL_PLC_Tests.Status.ActiveCaseId := 0;
    GVL_PLC_Tests.Status.ActiveCaseName := '';
    GVL_PLC_Tests.Status.ActiveStepId := 0;
    GVL_PLC_Tests.Status.ActiveStepName := '';
    GVL_PLC_Tests.Status.StepElapsed := T#0s;
    GVL_PLC_Tests.Status.StepTimeoutPT := T#0s;
END_IF;

// Agrégation globale des compteurs de cas de tests — seules les suites réellement
// exécutées CE run comptent (ChainMode = les deux ; sinon seule CurrentSuiteIdx)
// pour ne jamais compter les restes d'un run ciblé précédent sur l'autre suite.
PassedCount := 0;
FailedCount := 0;
TotalCount := 0;

IF ChainMode OR CurrentSuiteIdx = GVL_PLC_Tests_Const.SuiteSafety THEN
    FOR Idx := 1 TO GVL_PLC_Tests_Const.MaxTestCases DO
        IF instSafetyValidation.Report.Cases[Idx].Executed THEN
            TotalCount := TotalCount + 1;
            IF instSafetyValidation.Report.Cases[Idx].Ok THEN
                PassedCount := PassedCount + 1;
            ELSE
                FailedCount := FailedCount + 1;
            END_IF;
        END_IF;
    END_FOR;
END_IF;

IF ChainMode OR CurrentSuiteIdx = GVL_PLC_Tests_Const.SuiteTranslation THEN
    FOR Idx := 1 TO GVL_PLC_Tests_Const.MaxTestCases DO
        IF instTranslationValidation.Report.Cases[Idx].Executed THEN
            TotalCount := TotalCount + 1;
            IF instTranslationValidation.Report.Cases[Idx].Ok THEN
                PassedCount := PassedCount + 1;
            ELSE
                FailedCount := FailedCount + 1;
            END_IF;
        END_IF;
    END_FOR;
END_IF;

IF ChainMode OR CurrentSuiteIdx = GVL_PLC_Tests_Const.SuiteBucket THEN
    FOR Idx := 1 TO GVL_PLC_Tests_Const.MaxTestCases DO
        IF instBucketValidation.Report.Cases[Idx].Executed THEN
            TotalCount := TotalCount + 1;
            IF instBucketValidation.Report.Cases[Idx].Ok THEN
                PassedCount := PassedCount + 1;
            ELSE
                FailedCount := FailedCount + 1;
            END_IF;
        END_IF;
    END_FOR;
END_IF;

IF ChainMode OR CurrentSuiteIdx = GVL_PLC_Tests_Const.SuiteEncoder THEN
    FOR Idx := 1 TO GVL_PLC_Tests_Const.MaxTestCases DO
        IF instEncoderValidation.Report.Cases[Idx].Executed THEN
            TotalCount := TotalCount + 1;
            IF instEncoderValidation.Report.Cases[Idx].Ok THEN
                PassedCount := PassedCount + 1;
            ELSE
                FailedCount := FailedCount + 1;
            END_IF;
        END_IF;
    END_FOR;
END_IF;

IF ChainMode OR CurrentSuiteIdx = GVL_PLC_Tests_Const.SuiteModes THEN
    FOR Idx := 1 TO GVL_PLC_Tests_Const.MaxTestCases DO
        IF instModesValidation.Report.Cases[Idx].Executed THEN
            TotalCount := TotalCount + 1;
            IF instModesValidation.Report.Cases[Idx].Ok THEN
                PassedCount := PassedCount + 1;
            ELSE
                FailedCount := FailedCount + 1;
            END_IF;
        END_IF;
    END_FOR;
END_IF;

IF ChainMode OR CurrentSuiteIdx = GVL_PLC_Tests_Const.SuiteHeartbeat THEN
    FOR Idx := 1 TO GVL_PLC_Tests_Const.MaxTestCases DO
        IF instHeartbeatValidation.Report.Cases[Idx].Executed THEN
            TotalCount := TotalCount + 1;
            IF instHeartbeatValidation.Report.Cases[Idx].Ok THEN
                PassedCount := PassedCount + 1;
            ELSE
                FailedCount := FailedCount + 1;
            END_IF;
        END_IF;
    END_FOR;
END_IF;

GVL_PLC_Tests.Status.CasesTotal := TotalCount;
GVL_PLC_Tests.Status.CasesPassed := PassedCount;
GVL_PLC_Tests.Status.CasesFailed := FailedCount;

// 💓 Logique du Clignotant visuel d'activité (Heartbeat — Triple clignotement réactif)
IF GVL_PLC_Tests.Status.RunState = E_TestRunState.TESTRUN_RUNNING THEN
    // 1. Détection d'un changement de step réel -> Armement du triple clignotement
    IF GVL_PLC_Tests.Status.ActiveStepId <> LastStepId AND PulseCounter = 0 THEN
        PulseCounter := 1;
        CycleCounter := 0;
        GVL_PLC_Tests.Status.Heartbeat := TRUE;
        LastStepId := GVL_PLC_Tests.Status.ActiveStepId;
    END_IF;

    // 2. Gestion du cycle de clignotement (100ms ON / 100ms OFF x3)
    IF PulseCounter > 0 THEN
        CycleCounter := CycleCounter + 1;
        IF CycleCounter >= 10 THEN
            CycleCounter := 0;
            PulseCounter := PulseCounter + 1;
            IF PulseCounter <= 6 THEN
                // Impulsions impaires = TRUE, paires = FALSE
                GVL_PLC_Tests.Status.Heartbeat := (PulseCounter MOD 2 <> 0);
            ELSE
                // Fin du triple clignotement -> retour à l'état éteint
                PulseCounter := 0;
                GVL_PLC_Tests.Status.Heartbeat := FALSE;
            END_IF;
        END_IF;
    END_IF;
ELSE
    // Forcer à FALSE quand le runner est au repos
    GVL_PLC_Tests.Status.Heartbeat := FALSE;
    LastStepId := 0;
    PulseCounter := 0;
    CycleCounter := 0;
END_IF;
